PROGRAM MAIN
VAR
END_VAR

P_Tc3DALI_KL6821();

END_PROGRAM

(* stored: Version 1.1.0.1, ProductVersion 3.1.4024.0
   POU MAIN: Id {19621cf2-5ac2-4d67-acd2-73967a7641b8}, SpecialFunc None *)
